// TIA Portal V17 export
// export: Created 2022-07-20T06:59:48.6727059Z, ExportSetting WithDefaults, DisplayName Totally Integrated Automation Portal, DisplayVersion V17, DisplayName TIA Portal Openness, DisplayVersion V17, DisplayName TIA Portal Version Control Interface, DisplayVersion V17, DisplayName SINAMICS Startdrive Advanced, DisplayVersion V17, DisplayName SINAMICS Startdrive G130, G150, S120, S150, SINAMICS MV, S210, DisplayVersion V17, DisplayName SINAMICS Startdrive G110M, G120, G120C, G120D, G120P, G115D, DisplayVersion V17, DisplayName STEP 7 Professional, DisplayVersion V17, DisplayName STEP 7 Safety, DisplayVersion V17, DisplayName WinCC Advanced, DisplayVersion V17
FUNCTION_BLOCK "FB10221_SignalCounter"   // FB10221, LAD
TITLE = FB10221_SignalCounter
{ S7_Optimized_Access := 'TRUE' }
AUTHOR : Anirouddh
FAMILY : 1022x_COUNTERS
VERSION : 1.0
// Release note : 
// 1.0 - Feature developped
// stored: AutoNumber false, IsIECCheckEnabled false, IsRetainMemResEnabled false, MemoryReserve 100, SetENOAutomatically false, UDAEnableTagReadback false
   VAR_INPUT
      SignalToCount : Bool;
   END_VAR
   VAR_IN_OUT
      ResetCountner : Bool;
      SignalCounter : LReal;
   END_VAR
   VAR
      R_TRIG_SignalToCount : R_TRIG;
   END_VAR
BEGIN

REGION Network 1 (SCL): Edge Signals & Timers Manegement
   REGION EDGE SIGNALS
       #R_TRIG_SignalToCount(CLK := #SignalToCount);
   END_REGION
END_REGION

REGION Network 2 (SCL): Counter Management
   IF #R_TRIG_SignalToCount.Q THEN
       #SignalCounter += 1.0;
   ELSIF #ResetCountner THEN
       #SignalCounter := 0.0;
       IF #SignalCounter = 0.0 THEN
           #ResetCountner := FALSE;
       END_IF;
   END_IF;
END_REGION
END_FUNCTION_BLOCK
